// TwinCAT 3 PLC project PLC_Utilities
// ProgramVersion: 3.1.4024.0
// libraries:
//   Tc2_Standard, * (Beckhoff Automation GmbH)
//   Tc2_System, * (Beckhoff Automation GmbH)
//   Tc3_Module, * (Beckhoff Automation GmbH)
// project tree:
//   / PlcTask.TcTTO
//   POUs/ MAIN.TcPOU
// (motion and I/O tree: see PLC project plc1)
// real-time tasks:
//   TASK PlcTask: cycle T#10ms, priority 20, ADS port 350
//   TASK PlcTask1: cycle T#10ms, priority 21, ADS port 351

CONFIGURATION PLC_Utilities
    RESOURCE PLC ON TwinCAT3
        TASK PlcTask(INTERVAL := T#10ms, PRIORITY := 21);
        PROGRAM MAIN WITH PlcTask : MAIN;
    END_RESOURCE
END_CONFIGURATION

// ---- POUs/MAIN.TcPOU
PROGRAM MAIN
VAR

	out_warmup_state_sts 	AT %Q* 	: BYTE;
	out_activate_state_sts 	AT %Q* 	: BYTE;
	out_shutdown_state_sts 	AT %Q* 	: BYTE;
	out_error_sts			AT %Q*	: BOOL;
	out_error_code			AT %Q*	: DWORD;
	out_service1_sts		AT %Q*  : BYTE;
	out_service1_error_code AT %Q*	: DWORD;
	out_service2_sts		AT %Q*	: BYTE;
	out_service2_error_code AT %Q*	: DWORD;
	out_service3_sts		AT %Q*	: BYTE;
	out_service3_error_code AT %Q*	: DWORD;
	out_service4_sts		AT %Q*	: BYTE;
	out_service4_error_code AT %Q*	: DWORD;
	out_heartbeat			AT %Q* 	: BOOL;
	
END_VAR

END_PROGRAM
